Staubli VAL3: refresh.pgx

program refresh()
// page refresh
begin
  //
  // refresh the static message
  if (nKey>270 and nKey<=278) or (nKey==259 or nKey==264 or nKey==268) or use:bUseRefresh
    call refreshStatic()
    call refreshDynamic()
  else
    // refresh the Dynamic message
    if abs(clock()-nRefresh)>nTime
      call refreshDynamic()
    endIf
  endIf
end
